// Mitsubishi GX Works2 project: 램프   PLC: Q02/Q02H

PROGRAM MAIN
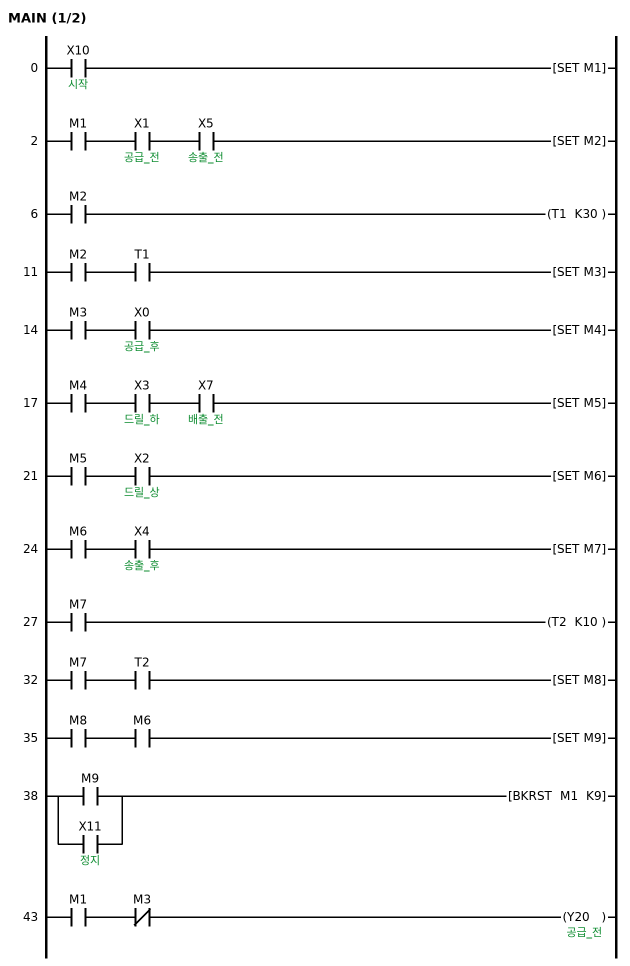
0     LD      X10  ; 시작
      SET     M1
2     LD      M1
      AND     X1  ; 공급_전
      AND     X5  ; 송출_전
      SET     M2
6     LD      M2
      OUT     T1 K30
11    LD      M2
      AND     T1
      SET     M3
14    LD      M3
      AND     X0  ; 공급_후
      SET     M4
17    LD      M4
      AND     X3  ; 드릴_하
      AND     X7  ; 배출_전
      SET     M5
21    LD      M5
      AND     X2  ; 드릴_상
      SET     M6
24    LD      M6
      AND     X4  ; 송출_후
      SET     M7
27    LD      M7
      OUT     T2 K10
32    LD      M7
      AND     T2
      SET     M8
35    LD      M8
      AND     M6
      SET     M9
38    LD      M9
      OR      X11  ; 정지
      BKRST   M1 K9
43    LD      M1
      ANI     M3
      OUT     Y20  ; 공급_전
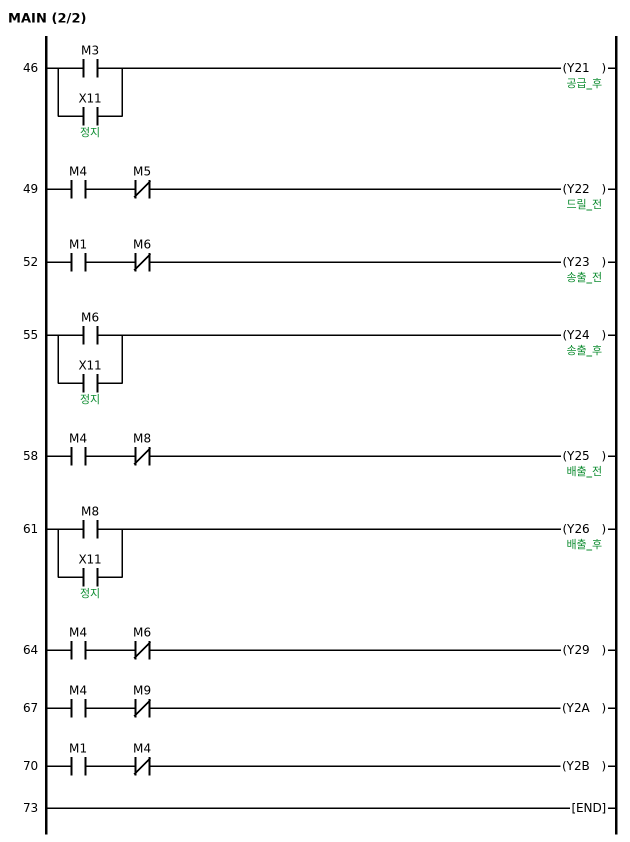
46    LD      M3
      OR      X11  ; 정지
      OUT     Y21  ; 공급_후
49    LD      M4
      ANI     M5
      OUT     Y22  ; 드릴_전
52    LD      M1
      ANI     M6
      OUT     Y23  ; 송출_전
55    LD      M6
      OR      X11  ; 정지
      OUT     Y24  ; 송출_후
58    LD      M4
      ANI     M8
      OUT     Y25  ; 배출_전
61    LD      M8
      OR      X11  ; 정지
      OUT     Y26  ; 배출_후
64    LD      M4
      ANI     M6
      OUT     Y29
67    LD      M4
      ANI     M9
      OUT     Y2A
70    LD      M1
      ANI     M4
      OUT     Y2B
73    END
END_PROGRAM

// device comments not shown above
X6  ; 배출_후
